# EPICS substitutions: ek9000App/Db/EL2001_mbboDirect.substitutions
file EL2001.template
{       pattern
        {
                TERMINAL,

        }
        {
        }
}
